Staubli VAL3: remEnableArm.pgx

program remEnableArm(string& sReturn[] (dimensions=1))
  local num nTimeout
begin
  // Turn arm power ON
  // Note that this will time out if you were not allowed to do it
  //
  logMsg("call remEnableArm")
  nTimeout=2
  if watch(nPPS>0,nTimeout)
    logMsg("PPS status ready for arm power.")
    if isPowered()==false
      enablePower()
    endIf
    if watch(isPowered(),nTimeout)
      sReturn="CMDENABLEARM"
      logMsg("Arm power ENABLED!")
      putln("Arm power ENABLED!")
    else

      if workingMode()!=4
        call remErrRemoteKey(sReturn)
      else
        call remErrTimeout(nTimeout,sReturn)
      endIf

    endIf


  else
    disablePower()
    call remErrPpTimeout(nTimeout,sReturn)
  endIf


end
